(* IEC 61131-3 sources: sps_maggio25/src/Lib, 4 files *)

(* ---- CustomTypes.st ---- *)
NAMESPACE Libreria.CustomTypes

    TYPE
        ValveState : INT (Opened := 1, Closed := 2, Error := 3, Undefined := 4) := Undefined;
    END_TYPE

END_NAMESPACE

(* ---- BasicValve.st ---- *)
NAMESPACE Libreria.Moduli

    FUNCTION BasicValve
        VAR_INPUT
            cmdOpen : BOOL;
        END_VAR

        VAR_OUTPUT
            ctrlOpen : BOOL;
        END_VAR

        ctrlOpen := cmdOpen;

    END_FUNCTION

    FUNCTION_BLOCK AdvancedValve
        VAR_INPUT
            cmdOpen : BOOL;
        END_VAR

        VAR_OUTPUT
            ctrlOpen : BOOL;
        END_VAR

        VAR
            isOpened : BOOL;
            isClosed : BOOL;
        END_VAR

        IF cmdOpen THEN
            ctrlOpen := TRUE;
            isOpened := TRUE;
            isClosed := FALSE;
        ELSE
            ctrlOpen := FALSE;
            isOpened := FALSE;
            isClosed := TRUE;
        END_IF;
    END_FUNCTION_BLOCK

END_NAMESPACE

(* ---- OOPValve.st ---- *)
USING Libreria.CustomTypes;
NAMESPACE Libreria.Moduli

    CLASS ClassValveBase
        VAR PUBLIC
            ctrlOpen : BOOL;
        END_VAR

        VAR
            isOpened : BOOL;
            isClosed : BOOL;
        END_VAR

        METHOD PUBLIC Open
            ctrlOpen := TRUE;
            isOpened := TRUE;
            isClosed := FALSE;
        END_METHOD

        METHOD PUBLIC Close
            ctrlOpen := FALSE;
            isOpened := FALSE;
            isClosed := TRUE;
        END_METHOD
    END_CLASS

    CLASS ClassValve
        VAR PUBLIC
            ctrlOpen : BOOL;
        END_VAR

        VAR
            actualState : ValveState;
        END_VAR

        METHOD PUBLIC Open
            ctrlOpen := TRUE;
            actualState := valveState#Opened;
        END_METHOD

        METHOD PUBLIC Close
            ctrlOpen := FALSE;
            actualState := valveState#Closed;
        END_METHOD

        METHOD PUBLIC GetState : ValveState;
            GetState := actualState;
        END_METHOD
    END_CLASS

    CLASS ClassValveBi EXTENDS ClassValve
        VAR PUBLIC
            //ctrlOpen : BOOL;      già presente in ClassValve!
            ctrlClose : BOOL;
        END_VAR

        METHOD PUBLIC OVERRIDE Open
            ctrlOpen := TRUE;
            ctrlClose := FALSE;
            actualState := valveState#Opened;
            END_METHOD

        METHOD PUBLIC OVERRIDE Close
            ctrlOpen := FALSE;
            ctrlClose := TRUE;
            actualState := valveState#Closed;
        END_METHOD

        // METHOD PUBLIC GetState          già presente in ClassValve!
    END_CLASS

END_NAMESPACE

(* ---- wrapperValve.st ---- *)
USING Libreria.CustomTypes;
NAMESPACE Libreria.Moduli

    FUNCTION_BLOCK WrapperValve

        VAR_INPUT
            wCmdOpen : BOOL;
        END_VAR

        VAR
            mainValve : ClassValve;
            actualState : ValveState;
        END_VAR

        VAR_OUTPUT
            wCtrlOpen : BOOL;
        END_VAR

        IF wCmdOpen THEN
            mainValve.Open();
        ELSE
            mainValve.Close();
        END_IF;

        wCtrlOpen := mainValve.ctrlOpen;
        actualState := mainValve.GetState();

    END_FUNCTION_BLOCK

END_NAMESPACE
